// Mitsubishi GX Works2 project: Termin4_Zadatak2   PLC: FX3S

// task Task_01 (event TRUE, interval 0, priority 31): POU_01

PROGRAM POU_01
VAR
  srednja_vrednost_1 : srednja_vrednost;
  temp1 : INT;
  temp2 : INT;
  rezultat : INT;
  klima_uredjaj_1 : klima_uredjaj;
  klima_uredjaj_2 : klima_uredjaj;
  grejac_klima1 : BOOL;
  grejac_klima2 : BOOL;
  senzori : INT;
  izlazi_tajmera : BOOL;
  TON_1 : TON;
  tajmer : TIME;
END_VAR
(* structured ladder/FBD written out as ST: instructions are called as NAME(EN, inputs, outputs); _pN, _eN, _tN stand for wires *)
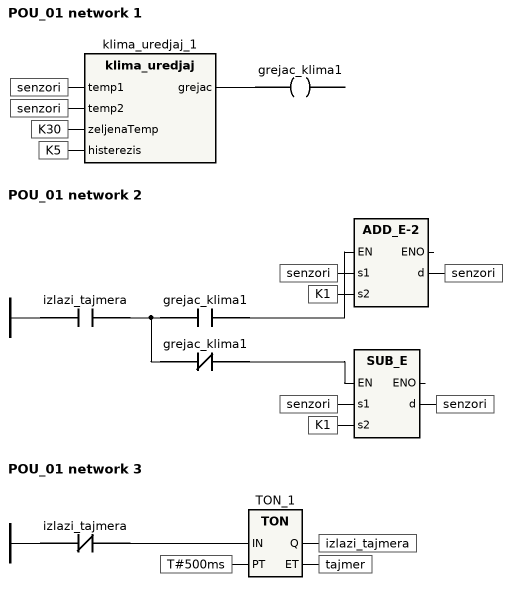
(* network 1 *)
klima_uredjaj_1(temp1 := senzori, temp2 := senzori, zeljenaTemp := K30, histerezis := K5);
grejac_klima1 := klima_uredjaj_1.grejac;
(* network 2 *)
ADD_E(izlazi_tajmera AND grejac_klima1, senzori, K1, senzori);
SUB_E(izlazi_tajmera AND NOT grejac_klima1, senzori, K1, senzori);
(* network 3 *)
TON_1(IN := NOT izlazi_tajmera, PT := T#500ms, Q => izlazi_tajmera, ET => tajmer);
END_PROGRAM

FUNCTION_BLOCK srednja_vrednost
VAR_INPUT
  temp_senzor1 : INT;
  temp_senzor2 : INT;
END_VAR
VAR
  zbir : INT;
END_VAR
VAR_OUTPUT
  srednja_vrednost : INT;
END_VAR
(* structured ladder/FBD written out as ST: instructions are called as NAME(EN, inputs, outputs); _pN, _eN, _tN stand for wires *)
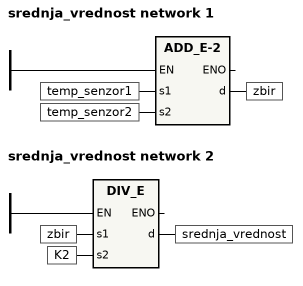
(* network 1 *)
ADD_E(TRUE, temp_senzor1, temp_senzor2, zbir);
(* network 2 *)
DIV_E(TRUE, zbir, K2, srednja_vrednost);
END_FUNCTION_BLOCK

FUNCTION_BLOCK klima_uredjaj
VAR
  srednja_vrednost_1 : srednja_vrednost;
END_VAR
VAR_INPUT
  temp1 : INT;
  temp2 : INT;
END_VAR
VAR
  trenutnaTemp : INT;
END_VAR
VAR_INPUT
  zeljenaTemp : INT;
  histerezis : INT;
END_VAR
VAR
  gornjiHisterezis : INT;
  donjiHisterezis : INT;
  stanje : ARRAY [0..2] OF BOOL;
END_VAR
VAR_OUTPUT
  grejac : BOOL;
END_VAR
VAR
  stanje_donje : ARRAY [0..2] OF BOOL;
END_VAR
(* structured ladder/FBD written out as ST: instructions are called as NAME(EN, inputs, outputs); _pN, _eN, _tN stand for wires *)
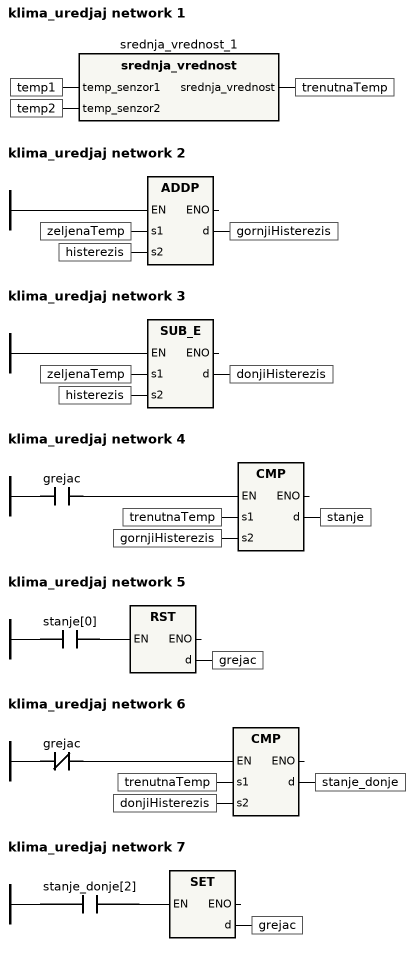
(* network 1 *)
srednja_vrednost_1(temp_senzor1 := temp1, temp_senzor2 := temp2, srednja_vrednost => trenutnaTemp);
(* network 2 *)
ADDP(TRUE, zeljenaTemp, histerezis, gornjiHisterezis);
(* network 3 *)
SUB_E(TRUE, zeljenaTemp, histerezis, donjiHisterezis);
(* network 4 *)
CMP(grejac, trenutnaTemp, gornjiHisterezis, stanje);
(* network 5 *)
RST(stanje[0], grejac);
(* network 6 *)
CMP(NOT grejac, trenutnaTemp, donjiHisterezis, stanje_donje);
(* network 7 *)
SET(stanje_donje[2], grejac);
END_FUNCTION_BLOCK
